// EXAMPLE: Customised FB_SENS_8_4 with additional User Configuration of channels
//          Only the M_UserConfigure() method is added to FB_SENS_8_4.
FUNCTION_BLOCK FB_SENS_8_4_USER_CONFIG EXTENDS FB_SENS_8_4
VAR_INPUT
END_VAR
VAR_OUTPUT
END_VAR
VAR
END_VAR

//
// Execute the base class FB_IODEV_SENS_8_4 object.
//
SUPER^();

// TODO_USER
//
// Define individual channel configurations, if used.
METHOD M_UserConfigure
VAR_INPUT
END_VAR
// TODO_USER
//
// Example implementation.
// Hard code any signal configuration.
//

// Configuration parameter cfg.bUserConfig defines if 
// the hard-coded configuration below should be used or
// the signals will be configured from the WS.

//
// Digital inputs
// Signal DI[0] is a LASER ON/OFF signal
// Signal DI[1] is a motor RUNNING/STOPPED signal
stat.arrDI[0].M_Configure('LASER OFF', 'LASER ON');
stat.arrDI[1].M_Configure('MOTOR STOPPED', 'MOTOR RUNNING');


//
// Analog inputs
//
stat.arrAI[0].M_Configure(CONVERSION_IODEV_NONE, 		0.0,   0.0, 0.0);
stat.arrAI[1].M_Configure(CONVERSION_IODEV_LINEAR, 		2.0,   1.0, 0.0);
stat.arrAI[2].M_Configure(CONVERSION_IODEV_QUADRATIC,	2.0,   1.0, 5.0);
// Edwards pressure guage
// P =10^(1.5*V - 12)    [mbar]
// 16-bit A/D converter, +=10V, e.g. EL3102.
// 1V = 2^16/10/2 = 3276.8 bit
// P = 10^(1.5*V - 12) = 10^(1.5/3276.8*bit - 12) = 10^(0.000457763*bit - 12)
stat.arrAI[3].M_Configure(CONVERSION_IODEV_EXP10, 	0.000457763, -12.0, 0.0);
END_METHOD

END_FUNCTION_BLOCK

(* stored: Version 1.1.0.1, ProductVersion 3.1.4022.16
   POU FB_SENS_8_4_USER_CONFIG: Id {dbf470de-1fa2-41a9-8c80-7ae28c2af164}, SpecialFunc None
   Method M_UserConfigure: Id {269945b5-dbf1-46f2-80fa-3bf3508f9ec0} *)
